// TIA Portal V15.1 export
// export: Created 2024-05-17T05:38:05.4670598Z, ExportSetting WithDefaults, DisplayName Totally Integrated Automation Portal, DisplayVersion V15.1 Update 5, DisplayName TIA Portal Openness, DisplayVersion V15.1 Update 5, DisplayName SINAMICS Startdrive Advanced, DisplayVersion V15.1, DisplayName G130, G150, S120, S150, SINAMICS MV, S210, DisplayVersion V15.1, DisplayName G110M, G120, G120C, G120D, G120P, DisplayVersion V15.1, DisplayName STEP 7 Professional, DisplayVersion V15.1 Update 5, DisplayName STEP 7 Safety, DisplayVersion V15.1, DisplayName WinCC Professional, DisplayVersion V15.1 Update 5, DisplayName SIMATIC Visualization Architect, DisplayVersion V15.1
ORGANIZATION_BLOCK "CYC_Proc"   // OB34, FBD, CyclicInterrupt
TITLE = CYC_Proc
{ S7_Optimized_Access := 'FALSE' }
VERSION : 0.1
// =============================================================================Cyclic Interrupt
// =============================================================================
// stored: AutoNumber false, IsIECCheckEnabled false, SetENOAutomatically False
   VAR_TEMP
      OB34_EV_CLASS : Byte;   // Bits 0-3 = 1 (Coming event), Bits 4-7 = 1 (Event class 1)
      OB34_STRT_INF : Byte;   // 16#35 (OB 34 has started)
      OB34_PRIORITY : Byte;   // Priority of OB Execution
      OB34_OB_NUMBR : Byte;   // 34 (Organization block 34, OB34)
      OB34_RESERVED_1 : Byte;   // Reserved for system
      OB34_RESERVED_2 : Byte;   // Reserved for system
      OB34_PHS_OFFSET : Int;   // Phase offset (integer, milliseconds)
      OB34_RESERVED_3 : Int;   // Reserved for system
      OB34_EXC_FREQ : Int;   // Frequency of execution (msec)
      OB34_DATE_TIME : Date_And_Time;   // Date and time OB34 started
   END_VAR
BEGIN

REGION Network 1: **** 1 - Inputs **** Incrementation of number of executions
   // Incrementation of number of executions
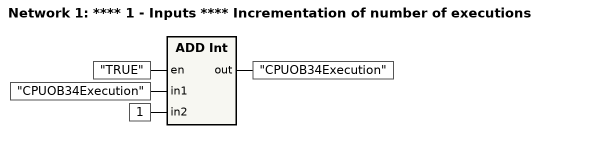
   IF "TRUE" THEN "CPUOB34Execution" := "CPUOB34Execution" + 1; END_IF;
END_REGION
END_ORGANIZATION_BLOCK
